FUNCTION_BLOCK UnitTestOnlyMismatchingNames EXTENDS FB_TestSuite

METHOD NameAlsoDoesntMatches
VAR_INPUT
END_VAR
TEST('This also doesnt match');

AssertTrue(Condition:=TRUE, Message:='Blabla');

TEST_FINISHED();
END_METHOD

METHOD NameDoesntMatch
TEST('This is completely different');

AssertTrue(Condition:=TRUE, Message:='Blabla');

TEST_FINISHED();
END_METHOD

END_FUNCTION_BLOCK

(* stored: Version 1.1.0.1, ProductVersion 3.1.4024.12
   POU UnitTestOnlyMismatchingNames: Id {b1c4a00b-5c5c-4336-a349-8d6258c04f41}, SpecialFunc None
   Method NameAlsoDoesntMatches: Id {6f280925-8f50-4f32-8fe1-54a2ccce582d}
   Method NameDoesntMatch: Id {c8bbb18e-2be6-4ff6-903b-8e71167a7a90} *)
